FUNCTION_BLOCK FB_Klep
VAR_INPUT
	i_eState 				: eSingleState;
	i_eModus				: eModus;
	i_eAutoWantedPosition 	: eValvePosition;
	i_eManualWantedPosition : eValvePosition;
	i_xHallSensorIn			: BOOL;
	i_xHallSensorOut 		: BOOL;
	i_xWarningReset			: BOOL;
	i_xAlarmReset			: BOOL;
END_VAR
VAR_OUTPUT
	o_eCurrentPosition 			: eValvePosition;
	o_xMagnetValve				: BOOL;
	o_xWarningPositionDown 		: BOOL; //Warning when position is down becease it not stopped the machineflow
	o_xErrorPositionUpOrUnknow	: BOOL; //Error when valve is up orunknow beceause it stopped te flow of the machine
	o_xAlarmPositionUpOrUnknow	: BOOL;
END_VAR
VAR
END_VAR

END_FUNCTION_BLOCK

(* stored: Version 1.1.0.1
   POU FB_Klep: Id {8f632325-bc23-4204-82f5-b4ed35cd42af}, SpecialFunc None *)
